(*
Casts I_Arg as I_RealArg
*)
FUNCTION ArgToIRealtArg : Result
VAR_INPUT
	iArg		: I_Arg;
END_VAR
VAR_OUTPUT
	iVal		: I_RealArg;
END_VAR

IF __QUERYINTERFACE(iArg, iVal) THEN
	ArgToIRealtArg := Ok;
END_IF

END_FUNCTION

(* stored: Version 1.1.0.1
   POU ArgToIRealtArg: Id {6990d5d4-7f95-460d-b805-d7b0f1d0f775}, SpecialFunc None *)
